FUNCTION_BLOCK FB_simulatiepompangout IMPLEMENTS ITF_pompangout

VAR
		internalState : int;
END_VAR

METHOD set : INT
VAR_INPUT
	state	: INT;
END_VAR
internalState := state;
END_METHOD

END_FUNCTION_BLOCK

(* stored: Version 1.1.0.1, ProductVersion 3.1.4026.8
   POU FB_simulatiepompangout: Id {4ca3763b-40d2-46a5-87ca-419448b32f65}, SpecialFunc None
   Method set: Id {3d4ff804-a469-4a9d-b82c-77714dc430b6} *)
